PROGRAM MAIN
VAR
END_VAR

//prg_Teleruptor();
//prg_Startveiligheid();
//prg_TrappenhuisautomaatVerlenging();
//prg_TrappenhuisautomaatTijdsinstelling();
//prg_Knipperlicht();
//prg_Millis();
//prg_OpenbaarToilet();
//prg_AutomatischeDeur();
//prg_Setpointsturing();
//prg_DraaiRichtingMotor();
//prg_Belsignaal();
//prg_Parking();
//prg_ProductenTellen();

END_PROGRAM

(* stored: Version 1.1.0.1, ProductVersion 3.1.4024.15
   POU MAIN: Id {ca3d6acd-d237-42df-a5f8-441aa260ece2}, SpecialFunc None *)
